PROGRAM MAIN
VAR
END_VAR

PrincipalClient();
PrincipalClient2();

END_PROGRAM

(* stored: Version 1.1.0.1, ProductVersion 3.1.4024.12
   POU MAIN: Id {3964b19e-6a02-4745-a8d7-adfb1df8383b}, SpecialFunc None *)
